(* PLC project Generated.project, CODESYS CODESYS V3.5 SP19 Patch 1 *)
(* stored: creationDateTime 2026-09-14T14:47:22.312065, modificationDateTime 2026-09-14T14:47:22.312065 *)

(* ======================================================================= ST_Modes_Autorisations - Bus public d'autorisations du mode machine ----------------------------------------------------------------------- Doc metier : DOC/AF/AF_Partie-05_Modes_Maintenance_v2.1.md DOC/AF/AF_Partie-02_Architecture_Programme_v3.2.md #2 NC-110 : le prefixe ST_fb* est reserve aux DUT propriete d'un seul FB. Ce DUT est un BUS multi-consommateurs (>=6 domaines : Cycle, Safety, Treuils, Translation, Supervision, Acquisition) -> renomme ST_Modes_Autorisations (bus de domaine public, sans le prefixe FB). Produit par FB_Modes (via PRG_03_Modes_Cycle) Consomme par : Cycle, Safety, Treuils, Translation, Supervision, Acquisition Producteur unique : FB_Modes (via PRG_03_Modes_Cycle) ======================================================================= *)
TYPE ST_Modes_Autorisations : STRUCT
  Mode : E_Mode;  (* Mode arbitre (DISABLE/N1/N2/SEMI_AUTO) *)
  SyncEnable : BOOL;  (* Synchro M1/M2 (logique positive) *)
  InhibitM1 : BOOL;  (* Inhibition M1 (MAINT_N2 only) *)
  InhibitM2 : BOOL;  (* Inhibition M2 (MAINT_N2 only) *)
  JoystickWinchSelectArbitrated : INT;  (* 0=M1+M2 couples nominal, 1=M1, 2=M2 (unitaires MAINT_N2) *)
  CoupledBucketPhaseLocked : BOOL;  (* T248 : phase mouvement couple VERROUILLEE pour ce maintien joystick -> la perte de l'etat ouvert/ferme en mouvement ne relance PAS de correction benne, ni de blocage "descente/montee interdite". Efface au relachement joystick confirme. *)
  WinchSelTransitionHold : BOOL;  (* T248 : changement de selecteur en cours -> requetes mouvement M1/M2 forcees a 0 jusqu'a l'arret confirme (pas de hand-off en mouvement) *)
  HomingApproachEnable : BOOL;  (* Depassement butee haut (N2) *)
  MaintenanceM3TargetEnable : BOOL;  (* Cible Translation Maintenance (N2 only) *)
  ModeChangePendingBlocked : BOOL;  (* AF-05 #4bis - matrice de maintenance Ces trois champs sont des FAITS/DIAGS publies, pas des autorisations : ils restent vrais meme quand le FB est neutralise par Enable=FALSE (etat persistant). Demande de changement de mode REFUSEE : les treuils *)
  ModeChangeBlockReason : STRING(40);  (* ne sont pas a l'arret mecanique confirme (contacteurs retombes ET frein serre ET |v| < seuil). Mode courant maintenu. Motif du blocage de bascule (texte IHM court, ex. "Chgt mode refuse : contacteur M1") *)
  M1ContactorsReleased : BOOL;  (* Détail des 6 sous-conditions de ModeChangeAllowed (diagnostic IHM) — TRUE = condition satisfaite. M1 : contacteurs retombés *)
  M1BrakeApplied : BOOL;  (* M1 : frein serré (NOT M1BrakeIsOpen) *)
  M1SpeedLow : BOOL;  (* M1 : vitesse sous seuil *)
  M2ContactorsReleased : BOOL;  (* M2 : contacteurs retombés *)
  M2BrakeApplied : BOOL;  (* M2 : frein serré (NOT M2BrakeIsOpen) *)
  M2SpeedLow : BOOL;  (* M2 : vitesse sous seuil *)
  HomingRequiredM1 : BOOL;  (* M1 : re-homing obligatoire avant tout retour SEMI_AUTO *)
  HomingRequiredM2 : BOOL;  (* M2 : idem *)
END_STRUCT;
END_TYPE

(* ======================================================================= 🪣 ST_ProgramBucketRequest — Demande de mouvement benne par le programme ─────────────────────────────────────────────────────────────── 🎯 Rôle : Regroupe les demandes logiques de manœuvre benne et mesure Kobold 📄 Référentiel : DOC/WFLOW/CONTRACTS/INTERPRG_CONTRACT_PRG03_MODES_CYCLE_v1.0.md ======================================================================= *)
TYPE ST_ProgramBucketRequest : STRUCT
  ReqOpen : BOOL;  (* Demande ouverture benne *)
  ReqClose : BOOL;  (* Demande fermeture benne *)
  ReqHoldAscentP1AfterClose : BOOL;  (* Maintien M2 en montee P1 apres fermeture, pour raccordement AX10B sans coupure *)
  ReqKoboldMeasureEnable : BOOL;  (* Demande activation mesure/contacteur Kobold *)
  DescendPermitDiveBucketOpen : BOOL;  (* Autorisation de descente conditionnée benne ouverte (DiveSearch) *)
  ExtractionControlActive : BOOL;  (* Plafond palier 1 pendant la montée contrôlée *)
  AscentPermit : BOOL;  (* Autorisation de remontée assistée (ExtractionAssist) *)
  MinStepDown : INT;  (* Palier plancher de descente imposé pendant la plongée (FB_DiveSearch, 0 = aucun) *)
END_STRUCT;
END_TYPE

(* ═══════════════════════════════════════════════════════════════ 🧩 ST_fbBucketCmdArbitration_Context — Contexte de gating benne ─────────────────────────────────────────────────────────────── 🎯 Rôle : Encapsuler les faits de gating consommés par FB_BucketCmdArbitration pour le séquencement couplé benne (config, intention both, état benne). Le FB dérive les flags armés (WinchBothDiveBucketOpenArmed / WinchBothAscentBucketCloseArmed) et les commandes arbitrées. 📤 Producteur : PRG_04_Treuils_Benne (câblage). 📄 Doc : DOC/AF/AF_Partie-10_Fonction_Winch_v2.1.md 🔌 État benne : 2 bits BOOL (BucketIsOpen/Closed) dérivés de _BucketState. ═══════════════════════════════════════════════════════════════ *)
TYPE ST_fbBucketCmdArbitration_Context : STRUCT
  TglEnableCoupledBucketSequencing : BOOL;  (* --> [CFG] Activation séquencement couplé benne (Commun.Cfg) *)
  MotionActive : BOOL;  (* --> [CMD] Intention mouvement both active (WinchBothMotionActive) *)
  ReqAscent : BOOL;  (* --> [CMD] Intention both montée *)
  ReqDescend : BOOL;  (* --> [CMD] Intention both descente *)
  BucketIsOpen : BOOL;  (* --> [STAT] Benne ouverte (BucketState.IsOpen) *)
  BucketIsClosed : BOOL;  (* --> [STAT] Benne fermée (BucketState.IsClosed) *)
  CoupledPhaseLocked : BOOL;  (* --> [STAT] T248 : phase couplée verrouillée (Auth.CoupledBucketPhaseLocked) -> ne PAS (ré)armer dive-open/ascent-close : plus de correction benne ni de blocage sur l'état temps réel une fois le mouvement lancé *)
END_STRUCT;
END_TYPE

(* ═══════════════════════════════════════════════════════════════ 🎛️ ST_fbBucketCmdArbitration_IHM — Entrées IHM de l'arbitrage benne ─────────────────────────────────────────────────────────────── 🎯 Rôle : Encapsuler les commandes IHM consommées par FB_BucketCmdArbitration (boutons ouverture/fermeture benne, nommage hardware propagé). 📤 Producteur : PRG_04_Treuils_Benne (câblage GVL_IHM). 📄 Doc : DOC/AF/AF_Partie-10_Fonction_Winch_v2.1.md 🔌 Nommage : BtnOpen/BtnClose = nommage hardware propagé (convention projet). ═══════════════════════════════════════════════════════════════ *)
TYPE ST_fbBucketCmdArbitration_IHM : STRUCT
  BtnOpen : BOOL;  (* --> [CMD] Bouton ouverture benne (M2TreuilBenne.Bucket.Cmd.BtnOpen) *)
  BtnClose : BOOL;  (* --> [CMD] Bouton fermeture benne (M2TreuilBenne.Bucket.Cmd.BtnClose) *)
END_STRUCT;
END_TYPE

(* values of E_Mode: DISABLE: Mode Désactivé / Veille de sécurité (sorties bloquées); MAINT_N1: Manuel Niveau 1 : Pilotage unitaire avec toutes sécurités actives; MAINT_N2: Manuel Niveau 2 : Pilotage dégradé (droits étendus + bypasses autorisés); SEMI_AUTO: Mode Semi-Automatique (séquenceur automatique) *)

{attribute 'qualified_only'}
{attribute 'strict'}
TYPE E_Mode : (DISABLE := 0, MAINT_N1 := 1, MAINT_N2 := 2, SEMI_AUTO := 3);
END_TYPE

(* ═══════════════════════════════════════════════════════════════ 🪣 FB_BucketCmdArbitration — Arbitrage de commande benne ─────────────────────────────────────────────────────────────── 🎯 Rôle : Arbitrer la source de commande benne (boutons IHM / séquencement couplé both / demande cycle selon le mode) et produire les commandes arbitrées (ouverture, fermeture, contacteur Kobold). 🔌 FB d'arbitrage (non-mouvement) : ne porte ni SafeStop ni StartStop de sécurité — il produit la commande logique, la safety reste dans FB_Bucket / FB_Safety_Winch. 📄 Doc : DOC/AF/AF_Partie-10_Fonction_Winch_v2.1.md 🔒 Bit-identique à l'ancien PRG_04 §1/§2 (refactor POO §5 : décision dans le FB, plus dans le PRG). Symétrique à FB_WinchCmdArbitrationM1/M2. ═══════════════════════════════════════════════════════════════ *)
FUNCTION_BLOCK FB_BucketCmdArbitration
  VAR_INPUT
    Enable : BOOL;  (* --> [CMD] Autorisation FB (TRUE=arbitre actif) *)
    Auth : ST_Modes_Autorisations;  (* --> [CMD] Autorisations mode (Mode, gating séquencement couplé) *)
    ReqBucket : ST_ProgramBucketRequest;  (* --> [REQ] Demande cycle benne (SEMI_AUTO) *)
    IHM : ST_fbBucketCmdArbitration_IHM;  (* --> [CMD] Boutons IHM benne (BtnOpen/BtnClose) *)
    Context : ST_fbBucketCmdArbitration_Context;  (* --> [STAT] Gating séquencement couplé benne *)
  END_VAR
  VAR_OUTPUT
    Ready : BOOL;  (* <-- [STAT] FB prêt à arbitrer (Enable) *)
    CmdOpen_IHM : BOOL;  (* <-- [CMD] Commande ouverture benne arbitrée *)
    CmdClose_IHM : BOOL;  (* <-- [CMD] Commande fermeture benne arbitrée *)
    KoboldContactorCmdArbitrated : BOOL;  (* <-- [CMD] Ordre contacteur capteur fond Kobold arbitré *)
    WinchBothDiveBucketOpenArmed : BOOL;  (* <-- [STAT] Séquencement couplé : descente benne ouverte armé *)
    WinchBothAscentBucketCloseArmed : BOOL;  (* <-- [STAT] Séquencement couplé : montée benne fermée armé *)
  END_VAR

            

// === IMPLEMENTATION ===

Ready := Enable;

IF NOT Enable THEN
    CmdOpen_IHM  := FALSE;
    CmdClose_IHM := FALSE;
    KoboldContactorCmdArbitrated := FALSE;
    WinchBothDiveBucketOpenArmed    := FALSE;
    WinchBothAscentBucketCloseArmed := FALSE;
ELSE
    // ── Règle absolue en pilotage both normal (bit-identique PRG_04 §1) ──
    // Descente autorisée UNIQUEMENT benne ouverte, montée UNIQUEMENT benne fermée.
    // T248 : une fois la phase couplée VERROUILLÉE (benne amenée dans l'état requis pour
    // ce maintien joystick), on n'arme plus dive-open / ascent-close -> la perte de
    // l'état ouvert/fermé EN MOUVEMENT ne relance aucune correction benne et ne bloque
    // plus le mouvement couplé ("descente/montée interdite" fantôme).
    WinchBothDiveBucketOpenArmed := Context.TglEnableCoupledBucketSequencing
        AND (Auth.Mode <> E_Mode.SEMI_AUTO)
        AND NOT Context.CoupledPhaseLocked
        AND Context.MotionActive AND Context.ReqDescend
        AND NOT Context.BucketIsOpen;
    WinchBothAscentBucketCloseArmed := Context.TglEnableCoupledBucketSequencing
        AND (Auth.Mode <> E_Mode.SEMI_AUTO)
        AND NOT Context.CoupledPhaseLocked
        AND Context.MotionActive AND Context.ReqAscent
        AND NOT Context.BucketIsClosed;

    // ── Ouverture benne : bouton IHM OU séquencement couplé descente benne ouverte
    //    OU demande cycle (bit-identique PRG_04 §2) ──
    CmdOpen_IHM := IHM.BtnOpen OR WinchBothDiveBucketOpenArmed OR ReqBucket.ReqOpen;

    // ── Fermeture benne : demande cycle > séquencement couplé montée benne fermée
    //    > bouton IHM (bit-identique PRG_04 §1) ──
    IF ReqBucket.ReqClose THEN
        CmdClose_IHM := TRUE;
    ELSIF WinchBothAscentBucketCloseArmed THEN
        CmdClose_IHM := TRUE;
    ELSE
        CmdClose_IHM := IHM.BtnClose;
    END_IF;

    // ── Contacteur Kobold : demande cycle (source unique PRG_03, bit-identique PRG_04 §1) ──
    KoboldContactorCmdArbitrated := ReqBucket.ReqKoboldMeasureEnable;
END_IF;

          
END_FUNCTION_BLOCK
